INTERFACE I_LinkedList EXTENDS I_Collection

METHOD PUBLIC AddAfter
VAR_INPUT
	After : I_LinkedListNode;
	Value : ANY;
END_VAR
END_METHOD

METHOD PUBLIC AddBefore
VAR_INPUT
	Before : I_LinkedListNode;
	Value : ANY;
END_VAR
END_METHOD

METHOD PUBLIC AddFirst
VAR_INPUT
	Value : ANY;
END_VAR
END_METHOD

METHOD PUBLIC AddLast
VAR_INPUT
	Value : ANY;
END_VAR
END_METHOD

METHOD PUBLIC Find : I_LinkedListNode
VAR_INPUT
	Value : ANY;
END_VAR
END_METHOD

METHOD PUBLIC FindLast : I_LinkedListNode
VAR_INPUT
	Value : ANY;
END_VAR
END_METHOD

PROPERTY PUBLIC First : I_LinkedListNode
GET
END_GET
END_PROPERTY

PROPERTY PUBLIC Last : I_LinkedListNode
GET
END_GET
END_PROPERTY

METHOD PUBLIC Remove
VAR_INPUT
	Value : ANY;
END_VAR
END_METHOD

METHOD PUBLIC RemoveFirst
END_METHOD

METHOD PUBLIC RemoveLast
END_METHOD

END_INTERFACE

(* stored: Version 1.1.0.1, ProductVersion 3.1.4024.12
   Itf I_LinkedList: Id {d65e86a0-7f4e-0ed4-1930-5fe7a71e95e5}
   Method AddAfter: Id {2028058f-b514-0af4-1fdd-424b77a21c18}
   Method AddBefore: Id {9c9bf288-4163-0c0b-326f-035f998eae45}
   Method AddFirst: Id {25e79b75-6a7b-0219-288f-38a1a515e787}
   Method AddLast: Id {4df6d425-8ae4-02d0-3964-645bf75862da}
   Method Find: Id {381e820c-6a05-06a4-102d-782a6a95b13b}
   Method FindLast: Id {0e27364e-c0cf-0134-034f-240b1bbe1576}
   Property First: Id {5deee7e8-e5f5-0d85-1f9c-97a893e0c28b}
   Get Get: Id {9fc5699c-b7e0-0f5f-1d8b-0f8588b8cb25}
   Property Last: Id {ee747e9f-3bbc-0f95-07e8-e10aeafa5136}
   Get Get: Id {b31b1324-2a9e-0d90-2b07-eaeca584e432}
   Method Remove: Id {81314fae-ae70-0bae-3069-787c7e6bfbfb}
   Method RemoveFirst: Id {3410b0c2-1774-0bdd-3e35-da68cf9f3bd8}
   Method RemoveLast: Id {ac44fde4-f603-0b74-1b5c-fa17e3478296} *)
